Fanuc KAREL source: kt00375.KL

-- PROVISIONAL review KL for V940-1; original PC SHA256 eb3c0401ade5b752a981d8ac90a0795cd230d904ceea4315eef8ec9f12a8c0ea
-- Incomplete behavior may be omitted. Consult companion uncertainty JSON. Do not deploy.
PROGRAM KT00375
%NOLOCKGROUP
VAR
  I2 : INTEGER
  OUT : BOOLEAN
-- UNRESOLVED_DECL Y1 type=002018
BEGIN
  -- V9_ZERO_TABLE_METADATA_HINT layout=0001; no indexed target words; source/name/runtime held
  -- UNRESOLVED_PC offsets 5-19; opcodes 2E,22,9D,33,B2
  -- UNRESOLVED_PC offsets 24-35; opcodes 2E,23
  -- UNRESOLVED_PC offsets 40-62; opcodes 22,9D,33,B1,21,5A,23
  -- UNRESOLVED_PC offsets 67-71; opcodes 7F
END KT00375
